{attribute addProperty BoxType "EPP6001-0002-0016"}
{attribute addProperty Id "COM_InputsAT %I*COM_Inputs_18212A5E192240COM_OutputsAT %Q*COM_Outputs_F536B385192240WcStateAT %I*WcState_F855686C1620InfoDataAT %I*InfoData_BC63D37F80100"}
{attribute addProperty CRC "1909685094"}
{attribute addProperty SizeInBites "480"}
{attribute addProperty SizeInBytes "60"}
TYPE EPP6001_4599C922 :
STRUCT
	{attribute addProperty Name "COM_Inputs"}
	COM_Inputs : COM_Inputs_18212A5E;
	{attribute addProperty Name "COM_Outputs"}
	COM_Outputs : COM_Outputs_F536B385;
	{attribute addProperty Name "WcState"}
	WcState : WcState_F855686C;
	{attribute addProperty Name "InfoData"}
	InfoData : InfoData_BC63D37F;
END_STRUCT
END_TYPE

(* stored: Version 1.2.0.0, ProductVersion 3.1.4024.9
   DUT EPP6001_4599C922: Id {619be79a-f404-4bae-91ae-52266ddeffb6} *)
